(* Schneider Machine Expert - Basic project TIMERS_ANALOG, file version 2.7.0.0 *)
(* ProjectInformations: Name=New project *)

HARDWARE
  Cpu 0: TM221CE16R
  ModuleExtensionObject 0: TM3AQ2/G
  EthernetConfiguration: NetworkName=M221, IpAllocationMode=FixedAddress, IpAddress=0.0.0.0, SubnetMask=0.0.0.0
  SerialLineConfiguration: Baud=Baud19200, Parity=ParityEven, DataBits=DataBits8, StopBits=StopBits1, PhysicalMedium=PhysicalMediumRs485, TransmissionMode=TransmissionModeModbusRtu, SlaveId=1, Addressing=SlaveAddressing
  MastTask: UsePeriodScanMode=false, PeriodScan=100
  FastTask: Period=255
  CpuBehavior: StartingMode=StartAsPreviousState, AutoSaveRamOnEeprom=true, WatchdogPeriod=250

SYMBOLS  (address, symbol, comment, settings)
  %TM0        [Preset=4, Base=OneSecond]
  %TM1        [Preset=8, Base=OneSecond]
  %I0.0     LOW_SPEED
  %I0.1     MID_SPEED
  %I0.2     HIGH_SPEED
  %IW0.0    SENSOR_01  [Type=Type_0_10V, Scope=Scope_Normal, Minimum=0, Maximum=1000]
  %QW1.0    VFD_SPEED  [Type=Type_0_10V, Scope=Scope_Customized, Minimum=0, Maximum=100]

POU New POU
  (* SectionNumber=1 *)

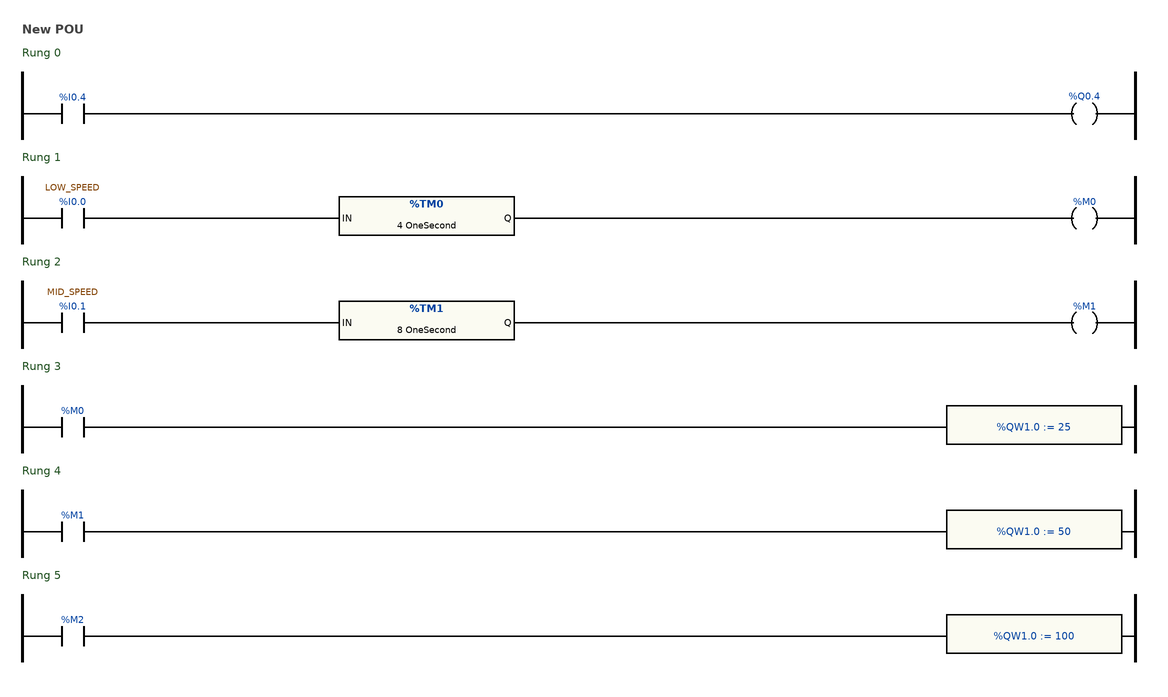

// Rung 0
  LD %I0.4
  ST %Q0.4
  // as ST:
  //   %Q0.4 := %I0.4;

// Rung 1
  BLK %TM0
  LD %I0.0                (* LOW_SPEED *)
  IN
  OUT_BLK
  LD Q
  ST %M0
  END_BLK
  // as ST:
  //   %TM0(IN := LOW_SPEED);
  //   %M0 := %TM0.Q;

// Rung 2
  BLK %TM1
  LD %I0.1                (* MID_SPEED *)
  IN
  OUT_BLK
  LD Q
  ST %M1
  END_BLK
  // as ST:
  //   %TM1(IN := MID_SPEED);
  //   %M1 := %TM1.Q;

// Rung 3
  LD %M0
  [ %QW1.0 := 25 ]        (* VFD_SPEED *)
  // as ST:
  //   IF %M0 THEN VFD_SPEED := 25; END_IF;

// Rung 4
  LD %M1
  [ %QW1.0 := 50 ]        (* VFD_SPEED *)
  // as ST:
  //   IF %M1 THEN VFD_SPEED := 50; END_IF;

// Rung 5
  LD %M2
  [ %QW1.0 := 100 ]       (* VFD_SPEED *)
  // as ST:
  //   IF %M2 THEN VFD_SPEED := 100; END_IF;
